RoboDK station: Test-Staubli.rdk

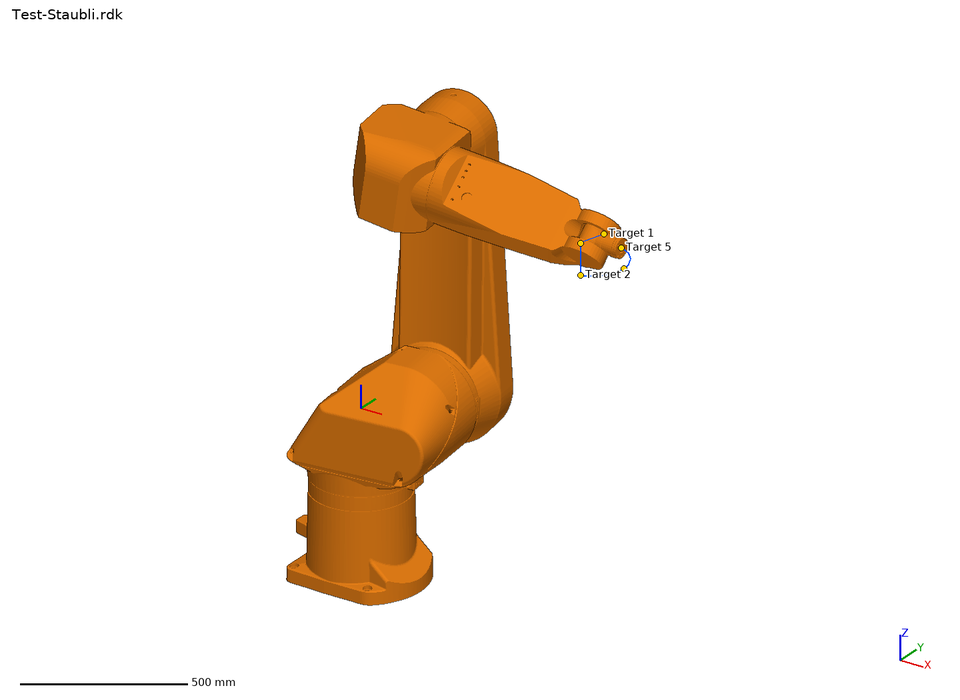
[picture v0: the station drawn from its stored meshes, robots at their saved joint values, targets as dots, program paths as lines]
Station staubli. Poses are relative to the parent item; angles as X-Y-Z fixed-axis rotations.
Station parameters (name, value as stored): IO_5, 1
  - frame Staubli RX160 Base at (0, 0, 550) mm
    - robot Staubli RX160: 6 axes, payload 20 kg, reach 1710 mm, repeatability 0.05 mm, weight 248 kg
        modified DH rows (alpha deg, a mm, theta deg, d mm): 0, 0, 0, 550; -90, 150, -90, 0; 0, 825, -90, 0; -90, 0, 0, 625; 90, 0, 0, 0; -90, 0, 180, 110
        base shift (0, 0, -550) mm
        joint limits [-160, -137.5, -150, -270, -105, -270] to [160, 137.5, 150, 270, 120, 270]; home [0, 0, 90, 0, 0, 0]; saved at [7.165, 0.593, 97.42, 222.045, 10.734, -221.543]
    - target Target 1 (Cartesian target) at (885, 0, 825) mm, rotated rx 0 ry 90 rz 0 deg; joints [0, 0, 90, 0, 0, 0] of Staubli RX160
    - target Target 2 (Cartesian target) at (885, -122.34, 737.83) mm, rotated rx 0 ry 90 rz 0 deg; joints [-8.971, 1.089, 96.914, 131.412, 12, -132.041] of Staubli RX160
    - target Target 3 (Cartesian target) at (885, -122.34, 843.05) mm, rotated rx 0 ry 90 rz 0 deg; joints [-8.971, 0.685, 87.654, 79.597, 9.122, -79.467] of Staubli RX160
    - target Target 4 (Cartesian target) at (966.62, -12.23, 737.83) mm, rotated rx 0 ry 90 rz 0 deg; joints [-0.818, 6.066, 91.523, 173.83, 7.633, -173.885] of Staubli RX160
    - target Target 5 (Cartesian target) at (881.36, 96.97, 737.83) mm, rotated rx 0 ry 90 rz 0 deg; joints [7.165, 0.593, 97.42, 222.045, 10.734, -221.543] of Staubli RX160
  - program Prog1 (13 instructions, listed below)
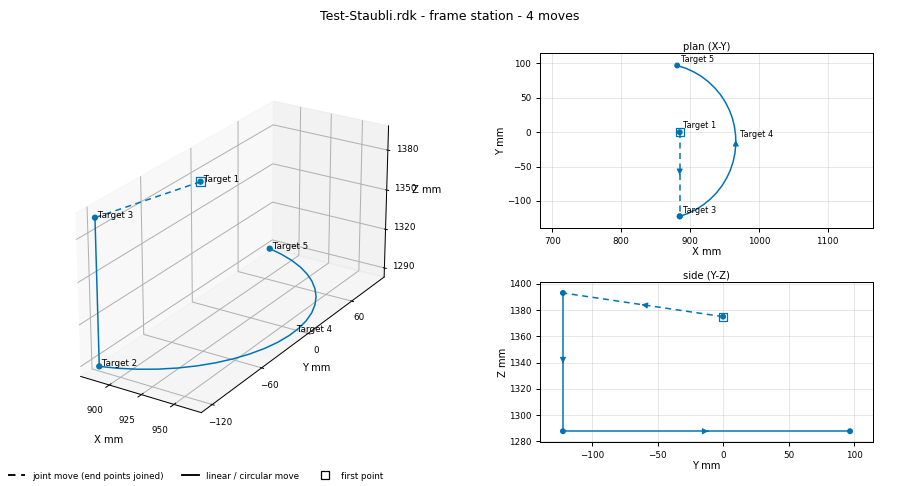
[picture p0: tool path of Test-Staubli.rdk in frame station, 4 of 4 moves have a stored position in this frame; points joined in program order, loops and branches not executed]

--- program Prog1 (robot Staubli RX160) ---
  Set Ref.: Staubli RX160 Base
  MoveJ (Target 1)
  MoveJ (Target 3)
  MoveL (Target 2)
  MoveC (Target 4, Target 5)
  Set speed (500.0 mm/s)
  Print: Display message
  Pause 500 ms
  Call Program1
  Set Ref.: Staubli RX160 Base
  Set Tool at (0, 0, 0) mm
  Set IO_5=1
  Wait IO_5=1 T5.0s
